FUNCTION_BLOCK AI_MUL_3 (* FB to calculate arithmetic MUL (generic FB) Adapter-Ausgang wird nur bei Wertänderung aktualisiert (Event nur bei tatsächlicher Änderung). *)
  (* Standard: 61131-3; Classification: standard arithmetic function; Description: Copyright (c) 2026 Meisterschulen am Ostbahnhof This program and the accompanying materials are made available under the terms of the Eclipse Public License 2.0 which is available at https://www.eclipse.org/legal/epl-2.0/ SPDX-License-Identifier: EPL-2.0 *)
  (* Version 1.0, 2026-04-20, Franz Höpfinger, Meisterschulen am Ostbahnhof, initial API and implementation and/or initial documentation *)
  PACKAGE adapter::iec61131::arithmetic;
  IMPORT eclipse4diac::core::GenericClassName;
  {SET_ATTRIBUTE(eclipse4diac::core::GenericClassName, 'GEN_AI_MUL')}
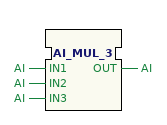
  SOCKETS
    IN1 : adapter::types::unidirectional::AI; (* MUL input 1 *)
    IN2 : adapter::types::unidirectional::AI; (* MUL input 2 *)
    IN3 : adapter::types::unidirectional::AI; (* MUL input 3 *)
  END_SOCKETS
  PLUGS
    OUT : adapter::types::unidirectional::AI; (* MUL result *)
  END_PLUGS
END_FUNCTION_BLOCK
